FUNCTION_BLOCK E_SWITCH_4 (* Switching (demultiplexing) an event based on boolean input G (4 channels, generic FB) *)
  (* Standard: 61499-1 Annex A; Classification: event function block; Function: Switching events (4 channels); Description: Copyright (c) 2017, 2026 fortiss GmbH, HR Agrartechnik GmbH This program and the accompanying materials are made available under the terms of the Eclipse Public License 2.0 which is available at https://www.eclipse.org/legal/epl-2.0/ SPDX-License-Identifier: EPL-2.0 Some portions generated by Gemini CLI *)
  (* Version 1.0, 2026-02-01, Franz Höpfinger, HR Agrartechnik GmbH, Initial creation based on E_SWITCH and E_SPLIT_3 *)
  PACKAGE iec61499::events;
  {SET_ATTRIBUTE(eclipse4diac::core::GenericClassName, 'GEN_E_SWITCH')}
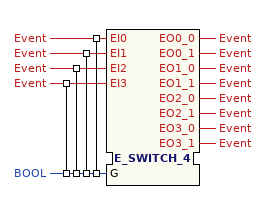
  EVENT_INPUT
    EI0 WITH G; (* Channel 0: Event Input *)
    EI1 WITH G; (* Channel 1: Event Input *)
    EI2 WITH G; (* Channel 2: Event Input *)
    EI3 WITH G; (* Channel 3: Event Input *)
  END_EVENT
  EVENT_OUTPUT
    EO0_0; (* Channel 0: Output, switched from EI0 when G=0 *)
    EO0_1; (* Channel 0: Output, switched from EI0 when G=1 *)
    EO1_0; (* Channel 1: Output, switched from EI1 when G=0 *)
    EO1_1; (* Channel 1: Output, switched from EI1 when G=1 *)
    EO2_0; (* Channel 2: Output, switched from EI2 when G=0 *)
    EO2_1; (* Channel 2: Output, switched from EI2 when G=1 *)
    EO3_0; (* Channel 3: Output, switched from EI3 when G=0 *)
    EO3_1; (* Channel 3: Output, switched from EI3 when G=1 *)
  END_EVENT
  VAR_INPUT
    G : BOOL; (* Channel 0-3: Switch EIn to EOn_0 when G=0, EIn to to EOn_1 when G=1 *)
  END_VAR
END_FUNCTION_BLOCK
